(* IEC 61131-3 sources: SRCI/RobotLibrary/RobotLibrary/POUs/AdvancedMove/MC_MoveLinearOffset, 1 file *)

(* ---- MC_MoveLinearOffsetFB.st ---- *)
/// Move the TCP relative to a reference cartesian position (linear interpolation)
FUNCTION_BLOCK MC_MoveLinearOffsetFB EXTENDS RobotLibraryBaseExecuteFB
// -------------------------------------------------------------------------
//  SRCI Robot Library
// -------------------------------------------------------------------------
//
//  Object:      MoveLinearOffsetFB
//  Author:      Thorsten Brach
//  Date:        2024-06-01
//
//  Description:
//
//
//  Copyright:
//    (C) 2024 Thorsten Brach. All rights reserved
//             Licensed under the LGPL-3.0 license.
//
//  Disclaimer:
//    This project is provided without any guarantee and can be used for
//    private and commercial purposes. Any use is at the user’s
//    own risk and responsibility.
//
// -------------------------------------------------------------------------
VAR_INPUT
  /// Parameter which determines the behavior towards the previously sent and still active or buffered commands
  AbortingMode       : AbortingMode;
  /// Defines the target sequence in which the command will be executed
  SequenceFlag       : SequenceFlag;
  /// command parameter
  ParCmd             : MoveLinearOffsetParCmd;
END_VAR

VAR_OUTPUT
  /// Command is transferred and confirmed by the RC
  CommandBuffered    : BOOL;
  /// The command takes control of the motion of the according axis group
  Active             : BOOL;
  /// The command was aborted by another command.
  CommandAborted     : BOOL;
  /// TRUE, while command is interrupted during execution and can be continued
  CommandInterrupted : BOOL;
  /// command outputs
  OutCmd             : MoveLinearOffsetOutCmd;
END_VAR

VAR
  /// internal copy of command parameter
 _parCmd             : MoveLinearOffsetParCmd;
  /// command data to send
 _command            : MoveLinearOffsetSendData;
  /// response data received
 _response           : MoveLinearOffsetRecvData;
END_VAR

  SUPER^(AxesGroup := AxesGroup);

END_FUNCTION_BLOCK

METHOD CheckParameterChanged : BOOL
VAR_IN_OUT
  /// Robot assignment of function
  AxesGroup    : AxesGroup;
END_VAR

  // Check ParCmd Size is > 0, becaue MemCmp does not work correctly with size = 0
  IF (SIZEOF(ParCmd) = 0)
  THEN
    RETURN;
  END_IF

  // compare memory
  CheckParameterChanged := ( MemCmp(ADR(ParCmd), ADR(_parCmd), SIZEOF(ParCmd)) <> RobotLibraryConstants.OK );

  IF ( CheckParameterChanged )
  THEN
    // update internal copy of parameters
   _parCmd := ParCmd;
    // inc parameter sequence
   _command.ParSeq := _command.ParSeq + 1;
    // update command data
    CommandData := CreateCommandPayload(); // ( Access via reference to rCommandFB in ACR )
    // notify active command register
    AxesGroup.Acyclic.ActiveCommandRegister.NotifyParameterChanged := _uniqueID;
  END_IF

END_METHOD

METHOD INTERNAL CreateCommandPayload : SendData
// Table 6-344: Sent CMD payload (PLC to RC) of "MoveLinearOffset"
// --------------------------
// Header
// --------------------------
// Byte 00 : UINT  - Type HB
// Byte 01 :       - Type LB
// Byte 02 : USINT - Reserve | ExecutionMode
// Byte 03 : USINT - ParSeq  | Priority
// --------------------------
// Datablock
// --------------------------
// Byte 04 : SINT  - EmitterID[0];
// Byte 05 : SINT  - EmitterID[1];
// Byte 06 : SINT  - EmitterID[2];
// Byte 07 : SINT  - EmitterID[3];
// Byte 08 : SINT  - ListenerID;
// Byte 09 : BYTE  - Reserved;
// Byte 10 : UINT  - VelocityRate HB;
// Byte 11 :       - VelocityRate LB;
// Byte 12 : UINT  - AccelerationRate HW HB;
// Byte 13 :       - AccelerationRate HW LB;
// Byte 14 : UINT  - DecelerationRate HW HB;
// Byte 15 :       - DecelerationRate HW LB;
// Byte 16 : UINT  - JerkRate HB;
// Byte 17 :       - JerkRate LB;
// Byte 18 : USINT - ToolNo;
// Byte 19 : USINT - FrameNo;
// Byte 20 : USINT - BlendingMode;
// Byte 21 : USINT - OriMode;
// Byte 22 : REAL  - BlendingParameter[0] HW HB;
// Byte 23 :       - BlendingParameter[0] HW LB;
// Byte 24 :       - BlendingParameter[0] LW HB;
// Byte 25 :       - BlendingParameter[0] LW LB;
// Byte 26 : REAL  - BlendingParameter[1] HW HB;
// Byte 27 :       - BlendingParameter[1] HW LB;
// Byte 28 :       - BlendingParameter[1] LW HB;
// Byte 29 :       - BlendingParameter[1] LW LB;
// Byte 30 : REAL  - ReferencePosition.X HW HB;
// Byte 31 :       - ReferencePosition.X HW LB;
// Byte 32 :       - ReferencePosition.X LW HB;
// Byte 33 :       - ReferencePosition.X LW LB;
// Byte 34 : REAL  - ReferencePosition.Y HW HB;
// Byte 35 :       - ReferencePosition.Y HW LB;
// Byte 36 :       - ReferencePosition.Y LW HB;
// Byte 37 :       - ReferencePosition.Y LW LB;
// Byte 38 : REAL  - ReferencePosition.Z HW HB;
// Byte 39 :       - ReferencePosition.Z HW LB;
// Byte 40 :       - ReferencePosition.Z LW HB;
// Byte 41 :       - ReferencePosition.Z LW LB;
// Byte 42 : REAL  - ReferencePosition.RX HW HB;
// Byte 43 :       - ReferencePosition.RX HW LB;
// Byte 44 :       - ReferencePosition.RX LW HB;
// Byte 45 :       - ReferencePosition.RX LW LB;
// Byte 46 : REAL  - ReferencePosition.RY HW HB;
// Byte 47 :       - ReferencePosition.RY HW LB;
// Byte 48 :       - ReferencePosition.RY LW HB;
// Byte 49 :       - ReferencePosition.RY LW LB;
// Byte 50 : REAL  - ReferencePosition.RZ HW HB;
// Byte 51 :       - ReferencePosition.RZ HW LB;
// Byte 52 :       - ReferencePosition.RZ LW HB;
// Byte 53 :       - ReferencePosition.RZ LW LB;
// Byte 54 : BYTE  - - - - - - W E S;
// Byte 55 : BYTE  - Reserved;
// Byte 56 : BYTE  - ReferencePosition.TurnNumber[0];
// Byte 57 : BYTE  - ReferencePosition.TurnNumber[1];
// Byte 58 : BYTE  - ReferencePosition.TurnNumber[2];
// Byte 59 : BYTE  - ReferencePosition.TurnNumber[3];
// Byte 60 : REAL  - ReferencePosition.E1 HW HB;
// Byte 61 :       - ReferencePosition.E1 HW LB;
// Byte 62 :       - ReferencePosition.E1 LW HB;
// Byte 63 :       - ReferencePosition.E1 LW LB;
// Byte 64 : REAL  - Offset.X HW HB;
// Byte 65 :       - Offset.X HW LB;
// Byte 66 :       - Offset.X LW HB;
// Byte 67 :       - Offset.X LW LB;
// Byte 68 : REAL  - Offset.Y HW HB;
// Byte 69 :       - Offset.Y HW LB;
// Byte 70 :       - Offset.Y LW HB;
// Byte 71 :       - Offset.Y LW LB;
// Byte 72 : REAL  - Offset.Z HW HB;
// Byte 73 :       - Offset.Z HW LB;
// Byte 74 :       - Offset.Z LW HB;
// Byte 75 :       - Offset.Z LW LB;
// Byte 76 : REAL  - Offset.RX HW HB;
// Byte 77 :       - Offset.RX HW LB;
// Byte 78 :       - Offset.RX LW HB;
// Byte 79 :       - Offset.RX LW LB;
// Byte 80 : REAL  - Offset.RY HW HB;
// Byte 81 :       - Offset.RY HW LB;
// Byte 82 :       - Offset.RY LW HB;
// Byte 83 :       - Offset.RY LW LB;
// Byte 84 : REAL  - Offset.RZ HW HB;
// Byte 85 :       - Offset.RZ HW LB;
// Byte 86 :       - Offset.RZ LW HB;
// Byte 87 :       - Offset.RZ LW LB;
// Byte 88 : BYTE  - - - - - - W E S;
// Byte 89 : BYTE  - Reserved;
// Byte 90 : BYTE  - Offset.TurnNumber[0];
// Byte 91 : BYTE  - Offset.TurnNumber[1];
// Byte 92 : BYTE  - Offset.TurnNumber[2];
// Byte 93 : BYTE  - Offset.TurnNumber[3];
// Byte 94 : REAL  - Offset.E1 HW HB;
// Byte 95 :       - Offset.E1 HW LB;
// Byte 96 :       - Offset.E1 LW HB;
// Byte 97 :       - Offset.E1 LW LB;
// Byte 98 : BOOL  - Manipulation;
// Byte 99 : BYTE  - Reserved;
// Byte 100: BYTE  - ConfigMode[0];
// Byte 101: BYTE  - ConfigMode[1];
// Byte 102: USINT - ReferenceType;
// Byte 103: USINT - TurnMode;
// Byte 104: UINT  - Time HB;
// Byte 105:       - Time LB;
// Byte 106: REAL  - ReferencePosition.E2 HW HB;
// Byte 107:       - ReferencePosition.E2 HW LB;
// Byte 108:       - ReferencePosition.E2 LW HB;
// Byte 109:       - ReferencePosition.E2 LW LB;
// Byte 110: REAL  - ReferencePosition.E3 HW HB;
// Byte 111:       - ReferencePosition.E3 HW LB;
// Byte 112:       - ReferencePosition.E3 LW HB;
// Byte 113:       - ReferencePosition.E3 LW LB;
// Byte 114: REAL  - ReferencePosition.E4 HW HB;
// Byte 115:       - ReferencePosition.E4 HW LB;
// Byte 116:       - ReferencePosition.E4 LW HB;
// Byte 117:       - ReferencePosition.E4 LW LB;
// Byte 118: REAL  - ReferencePosition.E5 HW HB;
// Byte 119:       - ReferencePosition.E5 HW LB;
// Byte 120:       - ReferencePosition.E5 LW HB;
// Byte 121:       - ReferencePosition.E5 LW LB;
// Byte 122: REAL  - ReferencePosition.E6 HW HB;
// Byte 123:       - ReferencePosition.E6 HW LB;
// Byte 124:       - ReferencePosition.E6 LW HB;
// Byte 125:       - ReferencePosition.E6 LW LB;
// Byte 126: REAL  - Offset.E2 HW HB;
// Byte 127:       - Offset.E2 HW LB;
// Byte 128:       - Offset.E2 LW HB;
// Byte 129:       - Offset.E2 LW LB;
// Byte 130: REAL  - Offset.E3 HW HB;
// Byte 131:       - Offset.E3 HW LB;
// Byte 132:       - Offset.E3 LW HB;
// Byte 133:       - Offset.E3 LW LB;
// Byte 134: REAL  - Offset.E4 HW HB;
// Byte 135:       - Offset.E4 HW LB;
// Byte 136:       - Offset.E4 LW HB;
// Byte 137:       - Offset.E4 LW LB;
// Byte 138: REAL  - Offset.E5 HW HB;
// Byte 139:       - Offset.E5 HW LB;
// Byte 140:       - Offset.E5 LW HB;
// Byte 141:       - Offset.E5 LW LB;
// Byte 142: REAL  - Offset.E6 HW HB;
// Byte 143:       - Offset.E6 HW LB;
// Byte 144:       - Offset.E6 LW HB;
// Byte 145:       - Offset.E6 LW LB;
// --------------------------

  // set command parameter
  _command.CmdTyp            :=  CmdType.MoveLinearOffset;
  _command.ExecMode          :=  ExecMode;
  _command.ParSeq            := _command.ParSeq;
  _command.Priority          :=  Priority;
  _command.EmitterID         := _parCmd.EmitterID;
  _command.Reserve           := 0;
  _command.ListenerID        := 0; {warning 'ToDo'}
  _command.Reserve           := 0;
  _command.VelocityRate      := REAL_TO_UINT(_parCmd.VelocityRate     * RobotLibraryConstants.REAL_CONVERSION_FACTOR);
  _command.AccelerationRate  := REAL_TO_UINT(_parCmd.AccelerationRate * RobotLibraryConstants.REAL_CONVERSION_FACTOR);
  _command.DecelerationRate  := REAL_TO_UINT(_parCmd.DecelerationRate * RobotLibraryConstants.REAL_CONVERSION_FACTOR);
  _command.JerkRate          := REAL_TO_UINT(_parCmd.JerkRate         * RobotLibraryConstants.REAL_CONVERSION_FACTOR);
  _command.ToolNo            := _parCmd.ToolNo;
  _command.FrameNo           := _parCmd.FrameNo;
  _command.BlendingMode      := _parCmd.BlendingMode;
  _command.OriMode           := _parCmd.OriMode;
  _command.BlendingParameter := _parCmd.BlendingParameter;
  _command.ReferencePosition := _parCmd.ReferencePosition;
  _command.Offset            := _parCmd.Offset;
  _command.Manipulation      := _parCmd.Manipulation;
  _command.Reserve2          := 0;
  _command.ConfigMode        := _parCmd.ConfigMode;
  _command.ReferenceType     := _parCmd.ReferenceType;
  _command.TurnMode          := _parCmd.TurnMode;
  _command.MoveTime          := TIME_TO_UINT(_parCmd.MoveTime);

  // copy command data to header
  _cmdHeader := _command;
  // call base implementation to copy header to payload buffer
  CreateCommandPayload := SUPER^.CreateCommandPayload();

  // add command.EmitterID[0]
  CreateCommandPayload.AddSint(_command.EmitterID[0]);
  // add command.EmitterID[1]
  CreateCommandPayload.AddSint(_command.EmitterID[1]);
  // add command.EmitterID[2]
  CreateCommandPayload.AddSint(_command.EmitterID[2]);
  // add command.EmitterID[3]
  CreateCommandPayload.AddSint(_command.EmitterID[3]);
  // add command.ListenerID
  CreateCommandPayload.AddSint(_command.ListenerID);
  // add command.Reserve
  CreateCommandPayload.AddByte(_command.Reserve);
  // add command.VelocityRate
  CreateCommandPayload.AddUint(_command.VelocityRate);
  // add command.AccelerationRate
  CreateCommandPayload.AddUint(_command.AccelerationRate);
  // add command.DecelerationRate
  CreateCommandPayload.AddUint(_command.DecelerationRate);
  // add command.JerkRate
  CreateCommandPayload.AddUint(_command.JerkRate);
  // add command.ToolNo
  CreateCommandPayload.AddUsint(_command.ToolNo);
  // add command.mFrameNo
  CreateCommandPayload.AddUsint(_command.FrameNo);
  // add command.BlendingMode
  CreateCommandPayload.AddUsint(_command.BlendingMode);
  // add command.OriMode
  CreateCommandPayload.AddUsint(_command.OriMode);
  // add command.BlendingParameter[0]
  CreateCommandPayload.AddReal(_command.BlendingParameter[0]);
  // add command.BlendingParameter[1]
  CreateCommandPayload.AddReal(_command.BlendingParameter[1]);
  // add command.ReferencePosition.X
  CreateCommandPayload.AddReal(_command.ReferencePosition.X);
  // add command.ReferencePosition.Y
  CreateCommandPayload.AddReal(_command.ReferencePosition.Y);
  // add command.ReferencePosition.Z
  CreateCommandPayload.AddReal(_command.ReferencePosition.Z);
  // add command.ReferencePosition.Rx
  CreateCommandPayload.AddReal(_command.ReferencePosition.Rx);
  // add command.ReferencePosition.Ry
  CreateCommandPayload.AddReal(_command.ReferencePosition.Ry);
  // add command.ReferencePosition.Rz
  CreateCommandPayload.AddReal(_command.ReferencePosition.Rz);
  // add command.ReferencePosition.Config
  CreateCommandPayload.AddArmConfig(_command.ReferencePosition.Config);
  // add command.ReferencePosition.TurnNumber
  CreateCommandPayload.AddTurnNumber(_command.ReferencePosition.TurnNumber);
  // add command.ReferencePosition.E1
  CreateCommandPayload.AddReal(_command.ReferencePosition.E1);
  // add command.Offset.X
  CreateCommandPayload.AddReal(_command.Offset.X);
  // add command.Offset.Y
  CreateCommandPayload.AddReal(_command.Offset.Y);
  // add command.Offset.Z
  CreateCommandPayload.AddReal(_command.Offset.Z);
  // add command.Offset.Rx
  CreateCommandPayload.AddReal(_command.Offset.Rx);
  // add command.Offset.Ry
  CreateCommandPayload.AddReal(_command.Offset.Ry);
  // add command.Offset.Rz
  CreateCommandPayload.AddReal(_command.Offset.Rz);
  // add command.Offset.Config
  CreateCommandPayload.AddArmConfig(_command.Offset.Config);
  // add command.Offset.TurnNumber
  CreateCommandPayload.AddTurnNumber(_command.Offset.TurnNumber);
  // add command.Offset.E1
  CreateCommandPayload.AddReal(_command.Offset.E1);
  // add command.Manipulation
  CreateCommandPayload.AddBool(_command.Manipulation);
  // add command.Reserve2
  CreateCommandPayload.AddByte(_command.Reserve2);
  // add command.ConfigMode
  CreateCommandPayload.AddArmConfig(_command.ConfigMode);
  // add command.ReferenceType
  CreateCommandPayload.AddUsint(_command.ReferenceType);
  // add command.TurnMode
  CreateCommandPayload.AddUsint(_command.TurnMode);
  // add command.MoveTime
  CreateCommandPayload.AddUint(_command.MoveTime);
  // add command.ReferencePosition.E2
  CreateCommandPayload.AddReal(_command.ReferencePosition.E2);
  // add command.ReferencePosition.E3
  CreateCommandPayload.AddReal(_command.ReferencePosition.E3);
  // add command.ReferencePosition.E4
  CreateCommandPayload.AddReal(_command.ReferencePosition.E4);
  // add command.ReferencePosition.E5
  CreateCommandPayload.AddReal(_command.ReferencePosition.E5);
  // add command.ReferencePosition.E6
  CreateCommandPayload.AddReal(_command.ReferencePosition.E6);
  // add command.Offset.E2
  CreateCommandPayload.AddReal(_command.Offset.E2);
  // add command.Offset.E3
  CreateCommandPayload.AddReal(_command.Offset.E3);
  // add command.Offset.E4
  CreateCommandPayload.AddReal(_command.Offset.E4);
  // add command.Offset.E5
  CreateCommandPayload.AddReal(_command.Offset.E5);
  // add command.Offset.E6
  CreateCommandPayload.AddReal(_command.Offset.E6);

END_METHOD

METHOD FB_init : BOOL
VAR_INPUT
  /// if TRUE, the retain variables are initialized (warm start / cold start)
	bInitRetains : BOOL;
  /// if TRUE, the instance afterwards gets moved into the copy code (online change)
	bInCopyCode  : BOOL;
END_VAR

  MyType := 'MC_MoveLinearOffsetFB';

END_METHOD

METHOD PROTECTED OnCall
VAR_IN_OUT
  /// Robot assignment of function
  AxesGroup : AxesGroup;
END_VAR

  // call base implementation
  SUPER^.OnCall(AxesGroup := AxesGroup);

  CASE _stepCmd OF

    00:  IF ( _execute_R.Q )
         THEN
           // set busy flag
           Busy := TRUE;
           // Reset command outputs
           MemSet(ADR(OutCmd),0,SIZEOF(OutCmd));
           // apply command parameter
          _parCmd := ParCmd;
           // init parameter sequence
          _command.ParSeq := 1;
           // set timeout
           SetTimeout(PT := _timeoutCmd, rTimer := _timerCmd);
           // inc step counter
          _stepCmd := _stepCmd + 1;
  	     END_IF

    01:  // create command data
         CommandData := CreateCommandPayload();
         // Add command to active command register
        _uniqueID := AxesGroup.Acyclic.ActiveCommandRegister.AddCmd( pCommandFB := ADR(THIS^ ));
         // set timeout
         SetTimeout(PT := _timeoutCmd, rTimer := _timerCmd);
         // inc step counter
        _stepCmd := _stepCmd + 1;

    02:  // Wait for responce received
         IF ( _responseReceived )
         THEN
           // reset response received flag
          _responseReceived := FALSE;
           // reset Active flag
           Active := FALSE;

           CASE  _response.State
           OF
             CmdMessageState.BUFFERED    : CommandBuffered    := TRUE;
             CmdMessageState.ACTIVE      : Active             := TRUE;
             CmdMessageState.INTERRUPTED : CommandInterrupted := TRUE;
             CmdMessageState.DONE        : Done               := TRUE;
             CmdMessageState.ABORTED     : CommandAborted     := TRUE;
             CmdMessageState.ERROR       : Error              := TRUE;
  				 END_CASE

           // Done, Aborted or Error ?
           IF (_response.State >= CmdMessageState.DONE )
           THEN
             // Reset Busy flag
             Busy := FALSE;
             // Update results
             OutCmd.Progress          := _response.Progress;
             OutCmd.FollowID          := _response.OriginID;
             OutCmd.RemainingDistance := _response.RemainingDistance;
             // set timeout
             SetTimeout(PT := _timeoutCmd, rTimer := _timerCmd);
             // inc step counter
            _stepCmd := _stepCmd + 1;
  				 END_IF
         END_IF

    03: IF ( NOT Execute)
        THEN
          Reset();
  			END_IF
  ELSE
    // invalid step
    ErrorID := RobotLibraryEvents.ERR_INVALID_STEP;
  END_CASE

  // Cancel
  IF (Busy) AND (NOT Execute)
  THEN
    // try to remove cmd
    AxesGroup.Acyclic.ActiveCommandRegister.RemoveCmd(_uniqueID);
  END_IF

  // Reset FB
  IF ( NOT Execute )
  THEN
    Reset();
  END_IF

END_METHOD

METHOD INTERNAL ParseResponsePayload : DINT
// Table 6-345: Received CMD payload (RC to PLC) of "MoveLinearOffset"
// --------------------------
// Header
// --------------------------
// Byte 00 : USINT   - ParSeq | State
// Byte 01 : SINT    - AlarmMessageSeverity
// Byte 02 : UINT    - AlarmMessageCode HB
// Byte 03 :         - AlarmMessageCode LB
// --------------------------
// Datablock
// --------------------------
// Byte 04 : USINT      - InvocationCounter
// Byte 05 : SINT       - Reserved
// Byte 06 : INT        - OriginID HB
// Byte 07 :            - OriginID LB
// Byte 08 : UINT       - Progress HB
// Byte 09 :            - Progress LB
// Byte 10 : REAL       - RemainingDistance HW HB
// Byte 11 :            - RemainingDistance HW LB
// Byte 12 :            - RemainingDistance LW HB
// Byte 13 :            - RemainingDistance LW LB
VAR_INPUT
  /// Response data
  ResponseData : RecvData;
END_VAR

  // call base implementation to parse the header from payload buffer
  ResponseData.PayloadPtr := SUPER^.ParseResponsePayload(ResponseData);

  // copy parsed header to response
  _response.ParSeq               := _rspHeader.ParSeq;
  _response.State                := _rspHeader.State;
  _response.AlarmMessageSeverity := _rspHeader.AlarmMessageSeverity;
  _response.AlarmMessageCode     := _rspHeader.AlarmMessageCode;

  // Get Response.InvocationCounter
  _response.InvocationCounter := ResponseData.GetUsint();
  // Get Response.Reserve
  _response.Reserve := ResponseData.GetSint();
  // Get Response.OriginID
  _response.OriginID := ResponseData.GetInt();
  // Get Response.Progress
  _response.Progress := ResponseData.GetUint();
  // Get Response.RemainingDistance
  _response.RemainingDistance := ResponseData.GetReal();

END_METHOD

METHOD PROTECTED Reset : DINT
VAR_INPUT
END_VAR

  Reset := SUPER^.Reset();

  Done               := FALSE;
  Busy               := FALSE;
  Active             := FALSE;
  CommandBuffered    := FALSE;
  CommandAborted     := FALSE;
  CommandInterrupted := FALSE;

END_METHOD
